// TIA Portal project "Pump_Faceplate_UDT" (V16)

(* hardware
DEVICE "S71500/ET200MP station_1"  S7-1500 station
   slot 0: "Rail_0"  Rack  6ES7 590-1***0-0AA0
   slot 0: "PM 70W 120/230VAC"  PM 70W 120/230VAC  6EP1332-4BA00
   slot 1: "PLC_1"  CPU 1511T-1 PN  6ES7 511-1TK01-0AB0  V2.8
      slot 3: "CPU display_1"  6ES7591-1AA00-0AA0
      slot 32768: "PROFINET interface_1"  X1
         slot 32769: "Port_1"  X1 P1
         slot 32770: "Port_2"  X1 P2
      slot 34817: "Virtual CP interface port_1"  Virtual CP interface port  Virtual CP interface port
   slot 2: "DI 16x24VDC BA_1"  DI 16x24VDC BA  6ES7 521-1BH10-0AA0  V1.1
   slot 3: "DQ 8x24VDC/2A HF_1"  DQ 8x24VDC/2A HF  6ES7 522-1BF00-0AB0  V2.2
   slot 4: "AI 4xU/I/RTD/TC ST_1"  AI 4xU/I/RTD/TC ST  6ES7 531-7QD00-0AB0  V1.0
   slot 5: "AQ 2xU/I ST_1"  AQ 2xU/I ST  6ES7 532-5NB00-0AB0  V1.0
DEVICE "HMI_1"  TP900 Comfort
   slot 0: "HMI_1"  TP900 Comfort  6AV2 124-0JC01-0AX0  16.0.0.0
   slot 1: "HMI_RT_1"  TP900 Comfort  6AV2 124-0JC01-0AX0  16.0.0.0
   slot 5: "HMI_1.IE_CP_1"  PROFINET Interface  16.0.0.0
      slot 1: "PROFINET Interface_1"  PROFINET Interface
         slot 1: "Port_1"  Port
         slot 2: "Port_2"  Port
   slot 7: "HMI_1.MPI/DP_CP_1"  MPI/DP Interface  16.0.0.0
*)

// ===== PLC "PLC_1"  CPU 1511T-1 PN =====

VAR_GLOBAL   // PLC tag table "Default tag table"
   "System_Byte" AT %MB1 : Byte;
   "FirstScan" AT %M1.0 : Bool;
   "DiagStatusUpdate" AT %M1.1 : Bool;
   "AlwaysTRUE" AT %M1.2 : Bool;
   "AlwaysFALSE" AT %M1.3 : Bool;
   "Clock_Byte" AT %MB0 : Byte;
   "Clock_10Hz" AT %M0.0 : Bool;
   "Clock_5Hz" AT %M0.1 : Bool;
   "Clock_2.5Hz" AT %M0.2 : Bool;
   "Clock_2Hz" AT %M0.3 : Bool;
   "Clock_1.25Hz" AT %M0.4 : Bool;
   "Clock_1Hz" AT %M0.5 : Bool;
   "Clock_0.625Hz" AT %M0.6 : Bool;
   "Clock_0.5Hz" AT %M0.7 : Bool;
   "Out_signal_mod" AT %MW2 : Int;
   "stop" AT %M4.0 : Bool;
   "signal_value" AT %MW6 : Int;
   "deviation_signal" AT %M8.0 : LReal;
END_VAR

TYPE "Pump_UDT"
   STRUCT
      bStart : Bool;
      bStop : Bool;
      bViev : Bool;
      iCurrent_level : Int;
   END_STRUCT;
END_TYPE

DATA_BLOCK "Pump_DB"   // DB1
{ S7_Optimized_Access := 'TRUE' }
VERSION : 0.1
   VAR
      Pump_HMI : "Pump_UDT";
      signal_DM : Array[0..20] of LReal;
      signal_int_DB : Array[0..20] of Int;
      start : Bool;
   END_VAR
BEGIN
   signal_DM[1] := 2.0;
   signal_DM[0] := 1.0;
   signal_DM[2] := 1.1;
   signal_DM[3] := 2.1;
   signal_DM[4] := 1.2;
   signal_DM[5] := 2.2;
   signal_DM[6] := 1.3;
   signal_DM[7] := 2.3;
   signal_DM[8] := 1.4;
   signal_DM[9] := 2.4;
   signal_DM[10] := 1.5;
   signal_DM[11] := 2.5;
   signal_DM[12] := 1.6;
   signal_DM[13] := 2.6;
   signal_DM[14] := 1.7;
   signal_DM[15] := 2.7;
   signal_DM[16] := 1.8;
   signal_DM[17] := 2.8;
   signal_DM[18] := 1.9;
   signal_DM[19] := 2.9;
   signal_DM[20] := 21.0;
   signal_int_DB[0] := 1;
   signal_int_DB[1] := 2;
   signal_int_DB[2] := 3;
   signal_int_DB[3] := 4;
   signal_int_DB[4] := 5;
   signal_int_DB[5] := 6;
   signal_int_DB[6] := 7;
   signal_int_DB[7] := 8;
   signal_int_DB[8] := 9;
   signal_int_DB[9] := 9;
   signal_int_DB[10] := 86;
   signal_int_DB[11] := 5;
   signal_int_DB[12] := 4;
END_DATA_BLOCK

DATA_BLOCK "Signal_modulation"   // DB2
{ S7_Optimized_Access := 'TRUE' }
VERSION : 0.1
   VAR
      Header : ArrayDBHeader;
      THIS : Array[0..20] of Int;
   END_VAR
BEGIN
   THIS[0] := 1;
   THIS[1] := 2;
   THIS[2] := 3;
   THIS[3] := 4;
   THIS[4] := 5;
   THIS[5] := 6;
   THIS[6] := 7;
   THIS[7] := 8;
   THIS[8] := 9;
   THIS[9] := 10;
   THIS[10] := 11;
   THIS[11] := 12;
   THIS[12] := 13;
   THIS[13] := 14;
   THIS[14] := 15;
   THIS[15] := 16;
   THIS[16] := 17;
   THIS[17] := 18;
   THIS[18] := 19;
   THIS[19] := 15;
   THIS[20] := 15;
   Header.LowerBound := 0;
   Header.UpperBound := 20;
   Header.Elements := 21;
   Header.PaddedSize := 2;
   Header.ElementSize := 2;
END_DATA_BLOCK

DATA_BLOCK "sensor_scale_DB"   // DB7
{ S7_Optimized_Access := 'TRUE' }
VERSION : 0.1
   VAR
      value : Array[0..5] of LReal;
   END_VAR
BEGIN
END_DATA_BLOCK

DATA_BLOCK "HMI_signal_db"   // DB8
{ S7_Optimized_Access := 'TRUE' }
VERSION : 0.1
   VAR
      HMI_signal_value : Int;
      HMI_signal_deviation : LReal;
   END_VAR
BEGIN
END_DATA_BLOCK

// folder: System blocks/Program resources

DATA_BLOCK "IEC_Counter_0_DB"   // DB3
{ S7_Optimized_Access := 'TRUE' }
AUTHOR : Simatic
FAMILY : IEC
NAME : CNTR
VERSION : 1.0
// stored: InstanceOfName IEC_COUNTER
"IEC_COUNTER"
BEGIN
END_DATA_BLOCK

DATA_BLOCK "ton1"   // DB4
{ S7_Optimized_Access := 'TRUE' }
AUTHOR : Simatic
FAMILY : IEC
NAME : IEC_TMR
VERSION : 1.0
// stored: InstanceOfName IEC_TIMER
"IEC_TIMER"
BEGIN
END_DATA_BLOCK

DATA_BLOCK "ton2"   // DB5
{ S7_Optimized_Access := 'TRUE' }
AUTHOR : Simatic
FAMILY : IEC
NAME : IEC_TMR
VERSION : 1.0
// stored: InstanceOfName IEC_TIMER
"IEC_TIMER"
BEGIN
END_DATA_BLOCK

DATA_BLOCK "ctu_count"   // DB6
{ S7_Optimized_Access := 'TRUE' }
AUTHOR : Simatic
FAMILY : IEC
NAME : CNTR
VERSION : 1.0
// stored: InstanceOfName IEC_COUNTER
"IEC_COUNTER"
BEGIN
END_DATA_BLOCK

// folder: (top level)

FUNCTION "Signal_modulation_FC" : Void   // FC1, SCL
{ S7_Optimized_Access := 'TRUE' }
VERSION : 0.1
   VAR_INPUT
      signal : Array[0..20] of Int;
   END_VAR
   VAR_OUTPUT
      Analog_out_signal : Int;
   END_VAR
   VAR_TEMP
      out_timer : Time;
      time_pt : S5Time;
      out_timer_pt : Bool;
      i : Int;
   END_VAR
BEGIN
END_FUNCTION

FUNCTION "secuense_array" : Void   // FC2, LAD
{ S7_Optimized_Access := 'TRUE' }
VERSION : 0.1
   VAR_INPUT
      input_sensor : Int;
      reset_scale : Bool;
   END_VAR
   VAR_OUTPUT
      out_array : Array[0..5] of LReal;
   END_VAR
   VAR_TEMP
      scale_sensor : LReal;
      index : Int;
      temp_lreal : LReal;
   END_VAR
BEGIN

REGION Network 1
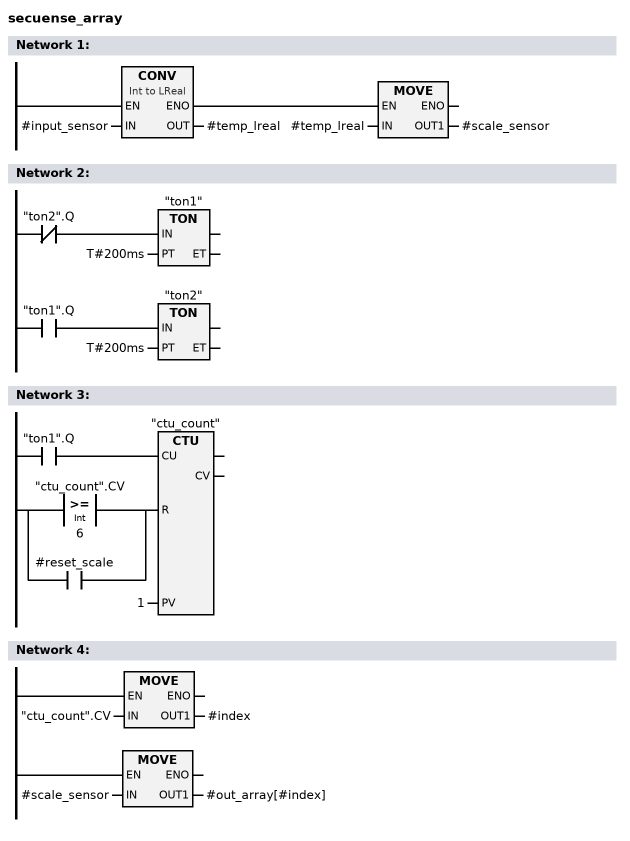
   RUNG wire#powerrail
      { S7_Templates := "[SrcType := Int, DestType := LReal]" } Convert(in := #input_sensor, out => #temp_lreal)
      Move(in := #temp_lreal, out1 => #scale_sensor)
   END_RUNG
   // the same network as SCL:
   #temp_lreal := INT_TO_LREAL(#input_sensor);
   #scale_sensor := #temp_lreal;
END_REGION

REGION Network 2
   "ton1".TON(IN := NOT "ton2".Q, PT := T#200ms);
   "ton2".TON(IN := "ton1".Q, PT := T#200ms);
END_REGION

REGION Network 3
   "ctu_count".CTU(CU := "ton1".Q, R := ("ctu_count".CV >= 6) OR #reset_scale, PV := 1);
END_REGION

REGION Network 4
   RUNG wire#powerrail
      Move(in := "ctu_count".CV, out1 => #index)
   END_RUNG
   RUNG wire#powerrail
      Move(in := #scale_sensor, out1 => #out_array[#index])
   END_RUNG
   // the same network as SCL:
   #index := "ctu_count".CV;
   #out_array[#index] := #scale_sensor;
END_REGION
END_FUNCTION

ORGANIZATION_BLOCK "Main"   // OB1, LAD, ProgramCycle
TITLE = "Main Program Sweep (Cycle)"
{ S7_Optimized_Access := 'TRUE' }
VERSION : 0.1
   VAR_INPUT
      Initial_Call : Bool;   // Initial call of this OB
      Remanence : Bool;   // =True, if remanent data are available
   END_VAR
   VAR_TEMP
      ret_val : Int;
      avg : LReal;
      devit : LReal;
      result : Int;
      up_integer : Int;
      reset : Bool;
   END_VAR
BEGIN

REGION Network 1
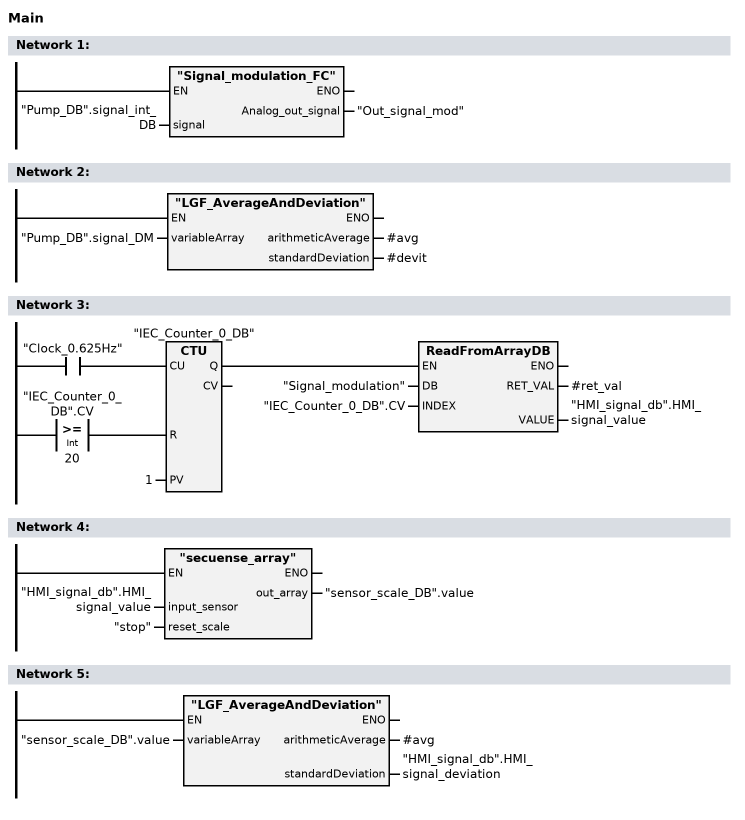
   RUNG wire#powerrail
      "Signal_modulation_FC"(signal := "Pump_DB".signal_int_DB, Analog_out_signal => "Out_signal_mod")
   END_RUNG
   // the same network as SCL:
   "Signal_modulation_FC"(signal := "Pump_DB".signal_int_DB, Analog_out_signal => "Out_signal_mod");
END_REGION

REGION Network 2
   RUNG wire#powerrail
      "LGF_AverageAndDeviation"(variableArray := "Pump_DB".signal_DM, arithmeticAverage => #avg, standardDeviation => #devit)
   END_RUNG
   // the same network as SCL:
   "LGF_AverageAndDeviation"(variableArray := "Pump_DB".signal_DM,
                           arithmeticAverage => #avg,
                           standardDeviation => #devit);
END_REGION

REGION Network 3
   // no SCL statement known for ReadFromArrayDB: written as a call
   "IEC_Counter_0_DB".CTU(CU := "Clock_0.625Hz", R := "IEC_Counter_0_DB".CV >= 20, PV := 1);
   IF "IEC_Counter_0_DB".Q THEN
       #ret_val := ReadFromArrayDB(db := "Signal_modulation",
                               index := "IEC_Counter_0_DB".CV,
                               value => "HMI_signal_db".HMI_signal_value);
   END_IF;
END_REGION

REGION Network 4
   RUNG wire#powerrail
      "secuense_array"(input_sensor := "HMI_signal_db".HMI_signal_value, reset_scale := "stop", out_array => "sensor_scale_DB".value)
   END_RUNG
   // the same network as SCL:
   "secuense_array"(input_sensor := "HMI_signal_db".HMI_signal_value,
                    reset_scale := "stop",
                    out_array => "sensor_scale_DB".value);
END_REGION

REGION Network 5
   RUNG wire#powerrail
      "LGF_AverageAndDeviation"(variableArray := "sensor_scale_DB".value, arithmeticAverage => #avg, standardDeviation => "HMI_signal_db".HMI_signal_deviation)
   END_RUNG
   // the same network as SCL:
   "LGF_AverageAndDeviation"(variableArray := "sensor_scale_DB".value,
                           arithmeticAverage => #avg,
                           standardDeviation => "HMI_signal_db".HMI_signal_deviation);
END_REGION
END_ORGANIZATION_BLOCK

// folder: LGF/9 Measurement operations

FUNCTION "LGF_AverageAndDeviation" : Void   // FC10006, SCL
TITLE = LGF_AverageAndDeviation
{ S7_Optimized_Access := 'TRUE' }
AUTHOR : Siemens_Digital_Industry
FAMILY : LGF
NAME : LGF_AverageAndDeviation
// This function calculates the arithmetic mean and the standard deviation from a series of numbers. / Diese Funktion berechnet aus einer Reihe von Zahlen das arithmetische Mittel und die Standardabweichung.
   VAR_INPUT
      variableArray : Array[*] of LReal;   // Sequence of numbers to calculate with / Zahlenreihe, mit der gerechnet werden soll
   END_VAR
   VAR_OUTPUT
      arithmeticAverage : LReal;   // Calculated arithmetic average value / Berechneter Arithmetischer Mittelwert
      standardDeviation : LReal;   // Calculated standard deviation / Berechnete Standardabweichung
   END_VAR
   VAR_TEMP
      tempLowerBound : Int;   // Temp lower bound
      tempUpperBound : Int;   // Temp upper bound
      tempNumberOfElements : Int;   // Temp number of elements
      tempSizeCounter : Int;   // Temp counter for loop
      tempArithmeticAverage : LReal;   // Temp calculated Arithmetic average
      tempStandardDeviation : LReal;   // Temp calculated Standard deviation
   END_VAR
   VAR CONSTANT
      NUMBER_OF_ELEMENTS_CORRECTION : Int := 1;   // Count also the starting value. e.g. [0.. 9] = 10 elements
      DIMENSION_ONE : UDInt := 1;   // First dimension of an array
      ZERO : LReal := 0.0;   // Initilization value
   END_VAR
BEGIN
   REGION Block info header
     //============================================================================
     // SIEMENS AG / (c)Copyright 2017
     //-----------------------------------------------------------------------------
     // Title:            LGF_AverageAndDeviation
     // Comment/Function: This function calculates the arithmetic average and the
     //                   standard deviation of a array of numbers
     // Library/Family:   LGF(Library General Functions)
     // Author:           Siemens Digital Industry Support
     // Tested with:      S7-PLCSIM Advanced V2.0 SP1
     // Engineering:      TIA Portal V15 Update 2
     // Restrictions:     ENO disabled - no error handling, ENO forced to true
     // Requirements:     PLC (S7-1200 / S7-1500)
     //------------------------------------------------------------------------------
     // Change log table:
     // Version  | Date       | Expert in charge       | Changes applied
     //----------|------------|------------------------|-----------------------------
     // 01.00.00 | 19.08.2015 | Siemens Industry Online Support
     //                       | First released version
     // 01.00.01 | 16.11.2015 | Siemens Industry Online Support
     //                       | Bug fix at WRONG_TYPE:  #error := true
     // 01.00.02 | 02.01.2017 | Siemens Industry Online Support
     //                       | Upgrade: TIA Portal V14 Update 1
     // 01.00.03 | 17.08.2018 | Siemens Industry Online Support
     //                       | Upgrade: TIA V15 Update 2
     // 01.00.04 | 23.11.2018 | Siemens Industry Online Support
     //                       | Upgrade: TIA V15.1
     // 02.00.00 | 25.01.2019 | Simatic Systems Support
     //                       | Data type changed from Variant to Array[*] of LReal
     // 02.00.01 | 31.10.2019 | Simatic Systems Support
     //                       | Regions, comments and constants are added
     // 03.00.00 | 23.04.2020 | Simatic Systems Support
     //                       | Set version to V3.0.0, harmonize the version of the whole library
     // 03.00.01 | 06.04.2021 | Simatic Systems Support
     //                       | Insert documentation
     //=============================================================================
   END_REGION Block info header

   REGION DESCRIPTION
     (/*An array of any size is connected via the `variableArray` input. After reading-out the array boundaries, the arithmetic mean value and the standard deviation will be calculated from the values and both will be output.

   ---

   Note
   :    An array with too many elements can cause the cycle monitoring time to be exceeded.
   Über den Eingang `variableArray` wird ein Array beliebiger Größe angeschlossen. Nach dem Auslesen der Array-Grenzen, wird aus den Werten der arithmetische Mittelwert und die Standardabweichung berechnet und beides ausgegeben.

   ---

   Hinweis
   :    Ein Array mit zu vielen Elementen kann zu einem Überschreiten der Zyklusüberwachungszeit führen.*/)
   END_REGION DESCRIPTION

   REGION Checking number of lower and upper bound
     #tempLowerBound := DINT_TO_INT(LOWER_BOUND(ARR := #variableArray, DIM := #DIMENSION_ONE));
     #tempUpperBound := DINT_TO_INT(UPPER_BOUND(ARR := #variableArray, DIM := #DIMENSION_ONE));

     // Upper - Lower bound gives the number of elements. +1 should be added for correct calculation.
     #tempNumberOfElements := #tempUpperBound - #tempLowerBound + #NUMBER_OF_ELEMENTS_CORRECTION;
   END_REGION

   REGION Calculation of the arithmetic average
     #tempArithmeticAverage := #ZERO;
     FOR #tempSizeCounter := #tempLowerBound TO #tempUpperBound DO
       #tempArithmeticAverage += #variableArray[#tempSizeCounter];
     END_FOR;

     #tempArithmeticAverage /= DINT_TO_REAL(#tempNumberOfElements);
   END_REGION

   REGION Calculation of the standard deviation
     #tempStandardDeviation := #ZERO;
     FOR #tempSizeCounter := #tempLowerBound TO #tempUpperBound DO
       #tempStandardDeviation += SQR((#variableArray[#tempSizeCounter] - #tempArithmeticAverage));
     END_FOR;

     #tempStandardDeviation := SQRT(#tempStandardDeviation / DINT_TO_REAL(#tempNumberOfElements));
   END_REGION

   REGION Writting to outputs
     #arithmeticAverage := #tempArithmeticAverage;
     #standardDeviation := #tempStandardDeviation;

     // ENO mechanism is not used - forced to true
     ENO := TRUE;
   END_REGION
END_FUNCTION

(* ===== HMI "HMI_RT_1" =====
system functions are stored by id; their names below are inferred from use
connection "HMI_Connection_1": ETHERNET, S7_1500_OMS

HMI tags "Default tag table"
   "Tag_ScreenNumber" : UInt, internal
   "signal_value" : Int = PLC signal_value AT %MW6, 1 s
   "deviation_signal" : LReal = PLC deviation_signal AT %M8.0, 1 s

HMI tags "Pump-HMI"
   "Pump_DB_Pump_HMI" : Pump_UDT = PLC Pump_DB.Pump_HMI, 1 s

HMI tags "HMI_signal"
   "HMI_signal_db_HMI_signal_value" : Int = PLC HMI_signal_db.HMI_signal_value, 1 s
   "HMI_signal_db_HMI_signal_deviation" : LReal = PLC HMI_signal_db.HMI_signal_deviation, 1 s

screen "Root screen" 800x420, template "Template_1"
   on GenerateScreen: SetTag("Tag_ScreenNumber", 1)
   SymbolLibrary "Symbol library_1" at 51,146 size 95x81
      on Activate: SetBit("bViev")
   ScreenModuleView "Pump_FP_1" at 5,2 size 141x133; ScreenModuleType ""
      Guid_{11997190-2812} <- "Pump_DB_Pump_HMI"
   TrendView "Trend view_1" at 151,0 size 633x356
   Button "Button_1" at 17,295 size 96x32; TextOff 'REFRESH'
      on Activate: ActivateScreen("Root screen", 0)

Template "Template_1" 800x420
   Button "Exit" at 720,360 size 78x58; TextOff 'Exit'; PictureOff "ExitRuntime_TP900_Comfort_TR"; PictureOn "ExitRuntime_TP900_Comfort_TR"
      on Release: StopRuntime(0)
   Button "Template_Button" at 640,360 size 78x58; TextOff 'Text'
   Button "Template_Button_1" at 560,360 size 78x58; TextOff 'Text'
   Button "Template_Button_2" at 480,360 size 78x58; TextOff 'Text'
   Button "Template_Button_3" at 400,360 size 78x58; TextOff 'Text'
   Button "Template_Button_4" at 321,360 size 78x58; TextOff 'Text'
   Button "Template_Button_5" at 241,360 size 78x58; TextOff 'Text'
   Button "Template_Button_6" at 161,360 size 78x58; TextOff 'Text'
   Button "Template_Button_7" at 81,360 size 78x58; TextOff 'Text'
   Button "Start screen" at 1,360 size 78x58; TextOff 'Start screen'; PictureOff "NavigateHome_TP900_Comfort_TR"; PictureOn "NavigateHome_TP900_Comfort_TR"
      on Release: ActivateScreen("Root screen", 0)
*)

(* ===== HMI "HMI_RT_1" =====

ScreenModuleEditorView "Pump_FP" 640x480
   IOField "I/O field_1" at 174,61 size 96x32; FormatPattern 99999
   Button "Button_1" at 174,141 size 96x32; TextOff 'Старт'
   Button "Button_2" at 29,141 size 96x32; TextOff 'Стоп'
   Button "Button_3" at 10,11 size 37x26; TextOff 'X'
   Button "Button_4" at 29,195 size 96x32; TextOff 'Управление'
   Button "Button_5" at 174,195 size 96x32; TextOff 'Авария'
   SymbolLibrary "Symbol library_1" at 41,57 size 84x66
*)

(* ===== HMI "HMI_RT_1" =====
system functions are stored by id; their names below are inferred from use

ScreenModuleEditorView "Pump_FP" 640x480
   Rectangle "Rectangle_1" at 10,10 size 279x247
      Visibility <- "fpPump.bViev"
   IOField "I/O field_1" at 174,61 size 96x32; FormatPattern 99999
      Visibility <- "fpPump.bViev"
   Button "Button_1" at 174,141 size 96x32; TextOff 'Старт'
      Visibility <- "fpPump.bViev"
   Button "Button_2" at 29,141 size 96x32; TextOff 'Стоп'
      Visibility <- "fpPump.bViev"
   Button "Button_3" at 10,11 size 37x26; TextOff 'X'
      Visibility <- "fpPump.bViev"
      on Press: ResetBit("fpPump.bViev")
   Button "Button_4" at 29,195 size 96x32; TextOff 'Управление'
      Visibility <- "fpPump.bViev"
   Button "Button_5" at 174,195 size 96x32; TextOff 'Авария'
      Visibility <- "fpPump.bViev"
   SymbolLibrary "Symbol library_1" at 41,57 size 84x66
      Visibility <- "fpPump.bViev"
*)